# EPICS SNL sequencer program: siteApps/SCL3Cooldown-sim-2-O/cooldownApp/src/CDOM036-1.stt
program CDOM0361Logic
option +r;

%% #include <math.h>

int om0361LogicProc[77];
assign om0361LogicProc to {
"SCL31-CDL01:VBx02-CV7301:CDLogic.PROC", "SCL31-CDL01:VBx04-CV7301:CDLogic.PROC", "SCL31-CDL01:VBx06-CV7301:CDLogic.PROC",
"SCL31-CDL01:VBx08-CV7301:CDLogic.PROC", "SCL31-CDL01:VBx10-CV7301:CDLogic.PROC", "SCL31-CDL01:VBx12-CV7301:CDLogic.PROC",
"SCL31-CDL01:VBx14-CV7301:CDLogic.PROC", "SCL31-CDL01:VBx16-CV7301:CDLogic.PROC", "SCL31-CDL01:VBx18-CV7301:CDLogic.PROC",
"SCL31-CDL01:VBx20-CV7301:CDLogic.PROC", "SCL31-CDL01:VBx22-CV7301:CDLogic.PROC", "SCL32-CDL02:VBx01-CV7301:CDLogic.PROC",
"SCL32-CDL02:VBx01-CV7201:CDLogic.PROC", "SCL32-CDL02:VBx02-CV7301:CDLogic.PROC", "SCL32-CDL02:VBx02-CV7201:CDLogic.PROC",
"SCL32-CDL02:VBx03-CV7301:CDLogic.PROC", "SCL32-CDL02:VBx03-CV7201:CDLogic.PROC", "SCL32-CDL02:VBx04-CV7301:CDLogic.PROC",
"SCL32-CDL02:VBx04-CV7201:CDLogic.PROC", "SCL32-CDL02:VBx05-CV7301:CDLogic.PROC", "SCL32-CDL02:VBx05-CV7201:CDLogic.PROC",
"SCL32-CDL02:VBx06-CV7301:CDLogic.PROC", "SCL32-CDL02:VBx06-CV7201:CDLogic.PROC", "SCL32-CDL02:VBx07-CV7301:CDLogic.PROC",
"SCL32-CDL02:VBx07-CV7201:CDLogic.PROC", "SCL32-CDL02:VBx08-CV7301:CDLogic.PROC", "SCL32-CDL02:VBx08-CV7201:CDLogic.PROC",
"SCL32-CDL02:VBx09-CV7301:CDLogic.PROC", "SCL32-CDL02:VBx09-CV7201:CDLogic.PROC", "SCL32-CDL02:VBx10-CV7301:CDLogic.PROC",
"SCL32-CDL02:VBx10-CV7201:CDLogic.PROC", "SCL32-CDL02:VBx11-CV7301:CDLogic.PROC", "SCL32-CDL02:VBx11-CV7201:CDLogic.PROC",
"SCL32-CDL02:VBx12-CV7301:CDLogic.PROC", "SCL32-CDL02:VBx12-CV7201:CDLogic.PROC", "SCL32-CDL02:VBx13-CV7301:CDLogic.PROC",
"SCL32-CDL02:VBx13-CV7201:CDLogic.PROC", "SCL32-CDL03:VBx01-CV7301:CDLogic.PROC", "SCL32-CDL03:VBx01-CV7201:CDLogic.PROC",
"SCL32-CDL03:VBx02-CV7301:CDLogic.PROC", "SCL32-CDL03:VBx02-CV7201:CDLogic.PROC", "SCL32-CDL03:VBx03-CV7301:CDLogic.PROC",
"SCL32-CDL03:VBx03-CV7201:CDLogic.PROC", "SCL32-CDL03:VBx04-CV7301:CDLogic.PROC", "SCL32-CDL03:VBx04-CV7201:CDLogic.PROC",
"SCL32-CDL03:VBx05-CV7301:CDLogic.PROC", "SCL32-CDL03:VBx05-CV7201:CDLogic.PROC", "SCL32-CDL03:VBx06-CV7301:CDLogic.PROC",
"SCL32-CDL03:VBx06-CV7201:CDLogic.PROC", "SCL32-CDL03:VBx07-CV7301:CDLogic.PROC", "SCL32-CDL03:VBx07-CV7201:CDLogic.PROC",
"SCL32-CDL03:VBx08-CV7301:CDLogic.PROC", "SCL32-CDL03:VBx08-CV7201:CDLogic.PROC", "SCL32-CDL03:VBx09-CV7301:CDLogic.PROC",
"SCL32-CDL03:VBx09-CV7201:CDLogic.PROC", "SCL32-CDL03:VBx10-CV7301:CDLogic.PROC", "SCL32-CDL03:VBx10-CV7201:CDLogic.PROC",
"SCL32-CDL03:VBx11-CV7301:CDLogic.PROC", "SCL32-CDL03:VBx11-CV7201:CDLogic.PROC", "SCL32-CDL03:VBx12-CV7301:CDLogic.PROC",
"SCL32-CDL03:VBx12-CV7201:CDLogic.PROC", "SCL32-CDL03:VBx13-CV7301:CDLogic.PROC", "SCL32-CDL03:VBx13-CV7201:CDLogic.PROC",
"SCL32-CDL03:VBx14-CV7301:CDLogic.PROC", "SCL32-CDL03:VBx14-CV7201:CDLogic.PROC", "SCL32-CDL03:VBx15-CV7301:CDLogic.PROC",
"SCL32-CDL03:VBx15-CV7201:CDLogic.PROC", "SCL32-CDL03:VBx16-CV7301:CDLogic.PROC", "SCL32-CDL03:VBx16-CV7201:CDLogic.PROC",
"SCL32-CDL03:VBx17-CV7301:CDLogic.PROC", "SCL32-CDL03:VBx17-CV7201:CDLogic.PROC", "SCL32-CDL03:VBx18-CV7301:CDLogic.PROC",
"SCL32-CDL03:VBx18-CV7201:CDLogic.PROC", "SCL32-CDL03:VBx19-CV7301:CDLogic.PROC", "SCL32-CDL03:VBx19-CV7201:CDLogic.PROC",
"P2DT-CDL04:VBx01-CV7301:CDLogic.PROC", "P2DT-CDL04:VBx01-CV7201:CDLogic.PROC"
};
monitor om0361LogicProc;

float valveVal[77];
assign valveVal to {
"SCL31-CDL01:VBx02-CV7301:Valve", "SCL31-CDL01:VBx04-CV7301:Valve", "SCL31-CDL01:VBx06-CV7301:Valve",
"SCL31-CDL01:VBx08-CV7301:Valve", "SCL31-CDL01:VBx10-CV7301:Valve", "SCL31-CDL01:VBx12-CV7301:Valve",
"SCL31-CDL01:VBx14-CV7301:Valve", "SCL31-CDL01:VBx16-CV7301:Valve", "SCL31-CDL01:VBx18-CV7301:Valve",
"SCL31-CDL01:VBx20-CV7301:Valve", "SCL31-CDL01:VBx22-CV7301:Valve", "SCL32-CDL02:VBx01-CV7301:Valve",
"SCL32-CDL02:VBx01-CV7201:Valve", "SCL32-CDL02:VBx02-CV7301:Valve", "SCL32-CDL02:VBx02-CV7201:Valve",
"SCL32-CDL02:VBx03-CV7301:Valve", "SCL32-CDL02:VBx03-CV7201:Valve", "SCL32-CDL02:VBx04-CV7301:Valve",
"SCL32-CDL02:VBx04-CV7201:Valve", "SCL32-CDL02:VBx05-CV7301:Valve", "SCL32-CDL02:VBx05-CV7201:Valve",
"SCL32-CDL02:VBx06-CV7301:Valve", "SCL32-CDL02:VBx06-CV7201:Valve", "SCL32-CDL02:VBx07-CV7301:Valve",
"SCL32-CDL02:VBx07-CV7201:Valve", "SCL32-CDL02:VBx08-CV7301:Valve", "SCL32-CDL02:VBx08-CV7201:Valve",
"SCL32-CDL02:VBx09-CV7301:Valve", "SCL32-CDL02:VBx09-CV7201:Valve", "SCL32-CDL02:VBx10-CV7301:Valve",
"SCL32-CDL02:VBx10-CV7201:Valve", "SCL32-CDL02:VBx11-CV7301:Valve", "SCL32-CDL02:VBx11-CV7201:Valve",
"SCL32-CDL02:VBx12-CV7301:Valve", "SCL32-CDL02:VBx12-CV7201:Valve", "SCL32-CDL02:VBx13-CV7301:Valve",
"SCL32-CDL02:VBx13-CV7201:Valve", "SCL32-CDL03:VBx01-CV7301:Valve", "SCL32-CDL03:VBx01-CV7201:Valve",
"SCL32-CDL03:VBx02-CV7301:Valve", "SCL32-CDL03:VBx02-CV7201:Valve", "SCL32-CDL03:VBx03-CV7301:Valve",
"SCL32-CDL03:VBx03-CV7201:Valve", "SCL32-CDL03:VBx04-CV7301:Valve", "SCL32-CDL03:VBx04-CV7201:Valve",
"SCL32-CDL03:VBx05-CV7301:Valve", "SCL32-CDL03:VBx05-CV7201:Valve", "SCL32-CDL03:VBx06-CV7301:Valve",
"SCL32-CDL03:VBx06-CV7201:Valve", "SCL32-CDL03:VBx07-CV7301:Valve", "SCL32-CDL03:VBx07-CV7201:Valve",
"SCL32-CDL03:VBx08-CV7301:Valve", "SCL32-CDL03:VBx08-CV7201:Valve", "SCL32-CDL03:VBx09-CV7301:Valve",
"SCL32-CDL03:VBx09-CV7201:Valve", "SCL32-CDL03:VBx10-CV7301:Valve", "SCL32-CDL03:VBx10-CV7201:Valve",
"SCL32-CDL03:VBx11-CV7301:Valve", "SCL32-CDL03:VBx11-CV7201:Valve", "SCL32-CDL03:VBx12-CV7301:Valve",
"SCL32-CDL03:VBx12-CV7201:Valve", "SCL32-CDL03:VBx13-CV7301:Valve", "SCL32-CDL03:VBx13-CV7201:Valve",
"SCL32-CDL03:VBx14-CV7301:Valve", "SCL32-CDL03:VBx14-CV7201:Valve", "SCL32-CDL03:VBx15-CV7301:Valve",
"SCL32-CDL03:VBx15-CV7201:Valve", "SCL32-CDL03:VBx16-CV7301:Valve", "SCL32-CDL03:VBx16-CV7201:Valve",
"SCL32-CDL03:VBx17-CV7301:Valve", "SCL32-CDL03:VBx17-CV7201:Valve", "SCL32-CDL03:VBx18-CV7301:Valve",
"SCL32-CDL03:VBx18-CV7201:Valve", "SCL32-CDL03:VBx19-CV7301:Valve", "SCL32-CDL03:VBx19-CV7201:Valve",
"P2DT-CDL04:VBx01-CV7301:Valve", "P2DT-CDL04:VBx01-CV7201:Valve"
};

monitor valveVal;

evflag  evFanout;
sync	valveVal	evFanout;

int index = 0;
assign index to "SCL3:CD-OM0361:IndexPV";
monitor index;

int proc = 1;

float om0361Val;
assign om0361Val to "SCL3:CD-OM0361:Value";
monitor om0361Val;

float cdDelay;
assign cdDelay to "SCL3:CD-OM0361:ScanTime";
monitor cdDelay;

float	valvewave[77];
assign	valvewave to "SCL3:CD-OM0361:ValveWave";
monitor valvewave;

ss ssCDOM0361
{
	state CDOM0361
	{
		when(delay(cdDelay))
		{
			if(om0361Val == 100) {
				om0361Val = 0;
				index++;
				pvPut(index, SYNC);
			} else {
				om0361Val = valveVal[index];
			};

			pvPut(om0361Val, SYNC);
			if(index < 77)
			{
				om0361LogicProc[index] = proc;
				pvPut(om0361LogicProc[index], SYNC);
			};
		}state CDOM0361
	}

}

ss ssOM0361ValveWave
{
	state init
	{
		when(TRUE)
		{
			efClear(evFanout);
		}state MakeOM0361ValveWave
	}

	state MakeOM0361ValveWave
	{
		when(efTestAndClear(evFanout))
		{
			int idx = 0;
			%%for(idx = 0; idx < 77;idx++)
				valvewave[idx] = valveVal[idx];

			pvPut(valvewave, SYNC);
		}state MakeOM0361ValveWave
	}
}
